FUNCTION Call_PositingBar

instControlBlockPositingBar(PartIsClamped := PositionerIsClamped,
							VerticalLimitReached := PositionerIsRaised,
							AlignmentDirection	:= PositingBarAlignmentDirection.AlingmentLeft,
							ActorInstanceIndex := 1,
							ActorInstanceName := '',
							OperatingMode := instOperatingMode.StateOperatingMode,
							HMIInterface := HMI.hmiMachineSectionInterface,
							Clamp => PositionerClamp,
							Raise =>PositionerRaise);
							
IF SimuClampPositingBar THEN
	SimuUnclampPositingBar := FALSE;
END_IF
IF SimuUnclampPositingBar THEN
	SimuClampPositingBar := FALSE;
END_IF
IF SimuRaisePositingBar THEN
	SimuLowerPositingBar := FALSE;
END_IF
IF SimuLowerPositingBar THEN
	SimuRaisePositingBar := FALSE;
END_IF

instControlBlockPositingBar.PositingBarClamping(SimuClampPositingBar);
instControlBlockPositingBar.PositingBarUnclamping(SimuUnclampPositingBar);
instControlBlockPositingBar.PositingBarRaise(SimuRaisePositingBar);
instControlBlockPositingBar.PositingBarLower(SimuLowerPositingBar);

END_FUNCTION

(* stored: Version 1.1.0.1
   POU Call_PositingBar: Id {371ad9e2-4cf0-498b-a263-772748bf8174}, SpecialFunc None *)
